FUNCTION_BLOCK FB_FeedForward
VAR_INPUT
	fXDotRef 	: LREAL; // Motion Referance
	fQMaxUp 	: LREAL; // Needs to be positive (22)
	fQMaxDown 	: LREAL; // Needs to be positive (15)
	fDeadUp		: LREAL; // Needs to be positive (0.155)
	fDeadDown 	: LREAL; // Needs to be positive (0.18)
END_VAR
VAR_OUTPUT
	fUFF : LREAL;
END_VAR
VAR
	fUTemp : LREAL;
	fUMax : LREAL := 0.9;
	fQRef : LREAL;
	fAp : LREAL := 33.1 / 10000.0;
	fAa : LREAL := 23.56 / 10000.0;
END_VAR


IF fXDotRef >= 0.0 THEN // Upwards
	
	fQRef := fAp * fXDotRef * 60000;
	fUTemp := -(fDeadUp + (fQRef/fQMaxUp) * (fUMax-fDeadUp));
	
//	IF fUTemp < -fUMax THEN
//		fUFF := -fUMax;
	
//	ELSIF fUTemp > -fDeadUp THEN
//		fUFF := -fDeadUp;
//	ELSE
//		fUFF := fUTemp;
//	END_IF

ELSIF fXDotRef < 0.0 THEN // Downwards
	
	fQRef := fAa * fXDotRef * 60000;
	fUTemp := -(-fDeadDown + (fQRef/fQMaxDown) * (fUMax-fDeadDown)); // FDeadDown needs to be positive
	
//	IF fUTemp > fUMax THEN
//		fUFF := fUMax;
	
//	ELSIF fUTemp < fDeadDown THEN
//		fUFF := fDeadDown;
//	ELSE
//		fUFF := fUTemp;
//	END_IF

END_IF

END_FUNCTION_BLOCK

(* stored: Version 1.1.0.1, ProductVersion 3.1.4024.12
   POU FB_FeedForward: Id {c7c6c1c3-721c-4ea2-9006-d66030d86044}, SpecialFunc None *)
